(* Logix 5000 project; controller AdvManLab vendor 1 type 14 code 158 rev 28.12; software revision 28.01 *)

TASK Festo (periodic, rate 50 ms, priority 10, watchdog 50 ms) : Data_Collection
TASK MainTask (continuous, watchdog 500 ms) : MainProgram
TASK SafetyTask (periodic, rate 20 ms, priority 10, watchdog 20 ms) : SafetyProgram

MODULES
   Local : vendor 1 type 14 code 158 (ICP 0, rev 28.12)
      EN2TR03 : vendor 1 type 12 code 200 (Ethernet 192.168.1.42, ICP 3, rev 5.8)
         CNC1 : vendor 1 type 14 code 178 (Ethernet 192.168.1.110, rev 28.1, $33999264$ RPI 10 ms)
         CNC4 : vendor 1 type 14 code 178 (Ethernet 192.168.1.140, rev 28.1, $0e99d22c$ RPI 10 ms)
         CNC3 : vendor 1 type 14 code 178 (Ethernet 192.168.1.130, rev 28.1, $2d1da0b6$ RPI 10 ms)
         CNC2 : vendor 1 type 14 code 178 (Ethernet 192.168.1.120, rev 28.1, $009657be$ RPI 10 ms)
      EN2TR02 : vendor 1 type 12 code 200 (ICP 2, Ethernet 192.168.1.41, rev 5.1)
         ConvETAP_N051 : 1783-ETAP (Ethernet 192.168.1.51, rev 2.2)
              Conv_N053:3:I.0   // C2 Entry RFID2
              Conv_N053:3:I.2   // C2 exit RFID4
              Conv_N053:3:I.1   // C1 Inside RFID3
              C3_N031:5:I.1   // C3 Outside RFID6
              C3_N031:5:I.0   // C3 Inside RFID5
              C2_N021:7:O.3   // CNC2_Switch_On
              C1_N011:6:I.7   // Inside C1 RFID1
              Main_N043:3:I.0   // C1 Entry NO RFID
         MainETAP_N044 : 1783-ETAP (Ethernet 192.168.1.44, rev 2.2)
         FanucLoopVFD_N045 : PowerFlex 525-EENET (Ethernet 192.168.1.45, rev 1.3, Output RPI 20 ms)
         ABBLoopVFD_N046 : PowerFlex 525-EENET (Ethernet 192.168.1.46, rev 1.3, Output RPI 20 ms)
         RFID_N057 : vendor 1 type 139 code 6 (Ethernet 192.168.1.57, rev 1.5, Output RPI 20 ms)
         RFID_N056 : vendor 1 type 139 code 6 (Ethernet 192.168.1.56, rev 1.5, Output RPI 20 ms)
              RFID_N056:I.Channel[0].TagPresent   // RFID5
              RFID_N056:I.Channel[1].TagPresent   // RFID6
         RFID_N054 : vendor 1 type 139 code 6 (Ethernet 192.168.1.54, rev 1.5, Output RPI 20 ms)
              RFID_N054:I.Channel[0].TagPresent   // RFID1
              RFID_N054:I.Channel[1].TagPresent   // RFID2
              RFID_N054:I.Channel[0].Data[3]   // Read tag Part #
              RFID_N054:I.Channel[0].Data[4]   // Read tag Process #
              RFID_N054:O.Channel[0].Data[3]   // Write Process #?
         RFID_N055 : vendor 1 type 139 code 6 (Ethernet 192.168.1.55, rev 1.5, Output RPI 20 ms)
              RFID_N055:I.Channel[0].TagPresent   // RFID3
              RFID_N055:I.Channel[1].TagPresent   // RFID4
         Fanuc_Rbt_C1 : ETHERNET-MODULE (Ethernet 192.168.1.12, rev 1.1, Output RPI 10 ms)
              Fanuc_Rbt_C1:I.Data[0].1   // Placement of part from CNC1 to conveyor Program finished DO[2]
              Fanuc_Rbt_C1:I.Data[0].0   // Placement of part from CNC2 to conveyor Program finished DO[1]
              Fanuc_Rbt_C1:I.Data[0].10   // Cell 1 Robot is at Hold Position (CNC2) DO[11]
              Fanuc_Rbt_C1:I.Data[0].11   // Robot has completed dropping off part (CNC2) DO[12]
              Fanuc_Rbt_C1:I.Data[0].12   // Robot has completed picking up part (CNC2) DO[13]
              Fanuc_Rbt_C1:I.Data[0].13   // Robot is dropping off part (CNC2) DO[14]
              Fanuc_Rbt_C1:I.Data[0].14   // Flip Part Program running DO[15]
              Fanuc_Rbt_C1:I.Data[0].15   // Flipping Part Program is Running DO[16]
              Fanuc_Rbt_C1:I.Data[0].2   // Pick from Conveyor and Drop on CNC2 Program running DO[3]
              Fanuc_Rbt_C1:I.Data[0].3   // Pick from Conveyor and Drop on CNC1 Program running DO[4]
              Fanuc_Rbt_C1:I.Data[0].4   // Pick from CNC2 and Drop on Conveyor Program running DO[5]
              Fanuc_Rbt_C1:I.Data[0].5   // Pick from CNC1 and Drop on Conveyor Program running DO[6]
              Fanuc_Rbt_C1:I.Data[0].6   // Cell 1 Robot is at Hold Position DI[7]
              Fanuc_Rbt_C1:I.Data[0].7   // Robot has completed dropping off part DI[8]
              Fanuc_Rbt_C1:I.Data[0].8   // Robot has completed picking up part DI[9]
              Fanuc_Rbt_C1:I.Data[0].9   // Robot is dropping off part DI[10]
              Fanuc_Rbt_C1:I.Data[1].0   // Pallet with Flipped Part can be Let Go DO[17]
              Fanuc_Rbt_C1:O.Data[0].0   // Pick from Conveyor and drop on CNC 2 DI[1]
              Fanuc_Rbt_C1:O.Data[0].1   // Pick from Conveyor and drop on CNC 1 DI[2]
              Fanuc_Rbt_C1:O.Data[0].2   // Pick from CNC2 and Drop on conveyor DI[3]
              Fanuc_Rbt_C1:O.Data[0].3   // Pick from CNC1 and Drop on conveyor DI[4]
              Fanuc_Rbt_C1:O.Data[0].4   // Flip part to machine top of cabin/trunk DI[5]
              Fanuc_Rbt_C1:O.Data[0].6   // Cell 1 Robot OK to Continue DI[7]
              Fanuc_Rbt_C1:O.Data[0].7   // Cell 2 Robot OK to Continue (CNC2) DI[8]
         Fanuc_Rbt_C2 : ETHERNET-MODULE (Ethernet 192.168.1.22, rev 1.1, Output RPI 8 ms)
              Fanuc_Rbt_C2:I.Data[0].10   // Cell 2 Robot is at Hold Position (CNC3) DO[11]
              Fanuc_Rbt_C2:I.Data[0].11   // Robot has completed dropping off part (CNC3) DO[12]
              Fanuc_Rbt_C2:I.Data[0].12   // Robot has completed picking up part (CNC3) DO[13]
              Fanuc_Rbt_C2:I.Data[0].13   // Robot is dropping off part (CNC3) DO[14]
              Fanuc_Rbt_C2:I.Data[0].2   // Pick from Conveyor and Drop on CNC3 Program running DO[3]
              Fanuc_Rbt_C2:I.Data[0].3   // Pick from Conveyor and Drop on CNC4 Program running DO[4]
              Fanuc_Rbt_C2:I.Data[0].4   // Pick from CNC3 and Drop on Conveyor Program running DO[5]
              Fanuc_Rbt_C2:I.Data[0].5   // Pick from CNC4 and Drop on Conveyor Program running DO[6]
              Fanuc_Rbt_C2:I.Data[0].6   // Cell 2 Robot is at Hold Position (CNC4) DO[7]
              Fanuc_Rbt_C2:I.Data[0].7   // Robot has completed dropping off part (CNC4) DO[8]
              Fanuc_Rbt_C2:I.Data[0].8   // Robot has completed picking up part (CNC4) DO[9]
              Fanuc_Rbt_C2:I.Data[0].9   // Robot is dropping off part (CNC4) DO[10]
              Fanuc_Rbt_C2:O.Data[0].0   // Pick from Conveyor and drop on CNC 3 DI[1]
              Fanuc_Rbt_C2:O.Data[0].1   // Pick from Conveyor and drop on CNC 4 DI[2]
              Fanuc_Rbt_C2:O.Data[0].2   // Pick from CNC3 and Drop on conveyor DI[3]
              Fanuc_Rbt_C2:O.Data[0].3   // Pick from CNC4 and Drop on conveyor DI[4]
              Fanuc_Rbt_C2:O.Data[0].6   // Cell 2 Robot OK to Continue (CNC4) DI[7]
              Fanuc_Rbt_C2:O.Data[0].7   // Cell 2 Robot OK to Continue (CNC3) DI[8]
              Fanuc_Rbt_C2:O.Data[1].0   // DI[17] Start
              Fanuc_Rbt_C2:O.Data[3].0   // DI[49]
              Fanuc_Rbt_C2:O.Data[3].1   // DI[50] Cycle Start / Run
              Fanuc_Rbt_C2:O.Data[3].2   // DI[51] Continue
              Fanuc_Rbt_C2:O.Data[3].8   // GI[1/0]
         Festo_CPX : ETHERNET-MODULE (Ethernet 192.168.1.245, rev 1.1, Output RPI 10 ms)
              Festo_CPX:I.Data[0]   // #0: FB36 - (I0)-LB
              Festo_CPX:I.Data[10]   // #5: 4AI-P-D10 - (I0)-LB
              Festo_CPX:I.Data[11]   // #5: 4AI-P-D10 - (I0)-HB
              Festo_CPX:I.Data[12]   // #5: 4AI-P-D10 - (I1)-LB
              Festo_CPX:I.Data[13]   // #5: 4AI-P-D10 - (I1)-HB
              Festo_CPX:I.Data[14]   // #5: 4AI-P-D10 - (I2)-LB
              Festo_CPX:I.Data[15]   // #5: 4AI-P-D10 - (I2)-HB
              Festo_CPX:I.Data[16]   // #5: 4AI-P-D10 - (I3)-LB
              Festo_CPX:I.Data[17]   // #5: 4AI-P-D10 - (I3)-HB
              Festo_CPX:I.Data[18]   // #6: MPA(S/F)-P - (I0)-LB
              Festo_CPX:I.Data[19]   // #6: MPA(S/F)-P - (I0)-HB
              Festo_CPX:I.Data[1]   // #0: FB36 - (I0)-HB
              Festo_CPX:I.Data[20]   // #3: 16DI-D - (I0-7)
              Festo_CPX:I.Data[21]   // #3: 16DI-D - (I8-15)
              Festo_CPX:I.Data[2]   // #1: 4AI-I - (I0)-LB
              Festo_CPX:I.Data[3]   // #1: 4AI-I - (I0)-HB
              Festo_CPX:I.Data[4]   // #1: 4AI-I - (I1)-LB
              Festo_CPX:I.Data[5]   // #1: 4AI-I - (I1)-HB
              Festo_CPX:I.Data[6]   // #1: 4AI-I - (I2)-LB
              Festo_CPX:I.Data[7]   // #1: 4AI-I - (I2)-HB
              Festo_CPX:I.Data[8]   // #1: 4AI-I - (I3)-LB
              Festo_CPX:I.Data[9]   // #1: 4AI-I - (I3)-HB
              Festo_CPX:O.Data[0]   // #0: FB36 - (O1)-LB
              Festo_CPX:O.Data[10]   // #10: MPA2S-D - (O0-3)
              Festo_CPX:O.Data[1]   // #0: FB36 - (O1)-HB
              Festo_CPX:O.Data[2]   // #2: 2AO - (O0)-LB
              Festo_CPX:O.Data[3]   // #2: 2AO - (O0)-HB
              Festo_CPX:O.Data[4]   // #2: 2AO - (O1)-LB
              Festo_CPX:O.Data[5]   // #2: 2AO - (O1)-HB
              Festo_CPX:O.Data[6]   // #4: 8DO - (O0-7)
              Festo_CPX:O.Data[7]   // #7: MPA2S-D - (O0-3)
              Festo_CPX:O.Data[8]   // #8: MPA2S-D - (O0-3)
              Festo_CPX:O.Data[9]   // #9: MPA2S-D - (O0-3)
              Festo_CPX:C.Data[113].0   // -
              Festo_CPX:C.Data[144].7   // -
              Festo_CPX:C.Data[28].7   // -
              Festo_CPX:C.Data[2].7   // -
              Festo_CPX:C.Data[53].0   // -
              Festo_CPX:C.Data[53].2   // -
              Festo_CPX:C.Data[53].3   // -
              Festo_CPX:C.Data[53].4   // -
              Festo_CPX:C.Data[53].5   // -
              Festo_CPX:C.Data[53].6   // -
              Festo_CPX:C.Data[54].0   // -
              Festo_CPX:C.Data[54].2   // -
              Festo_CPX:C.Data[54].4   // -
              Festo_CPX:C.Data[113].1   // -
              Festo_CPX:C.Data[113].2   // -
              Festo_CPX:C.Data[54].5   // -
              Festo_CPX:C.Data[54].6   // -
              Festo_CPX:C.Data[54].7   // -
              Festo_CPX:C.Data[55].0   // -
              Festo_CPX:C.Data[55].1   // -
              Festo_CPX:C.Data[55].2   // -
              Festo_CPX:C.Data[55].3   // -
              Festo_CPX:C.Data[55].6   // -
              Festo_CPX:C.Data[55].7   // -
              Festo_CPX:C.Data[67].4   // -
              Festo_CPX:C.Data[67].5   // -
              Festo_CPX:C.Data[113].3   // -
              Festo_CPX:C.Data[113].4   // -
              Festo_CPX:C.Data[113].5   // -
              Festo_CPX:C.Data[1].7   // -
              Festo_CPX:C.Data[21].2   // -
              Festo_CPX:C.Data[21].3   // -
              Festo_CPX:C.Data[21].4   // -
              Festo_CPX:C.Data[21].5   // -
              Festo_CPX:C.Data[113].6   // -
              Festo_CPX:C.Data[128].1   // O0: Failsafe - Bit1
              Festo_CPX:C.Data[67].6   // -
              Festo_CPX:C.Data[67].7   // -
              Festo_CPX:C.Data[74].1   // -
              Festo_CPX:C.Data[74].2   // -
              Festo_CPX:C.Data[74].3   // -
              Festo_CPX:C.Data[74].4   // -
              Festo_CPX:C.Data[74].5   // -
              Festo_CPX:C.Data[74].6   // -
              Festo_CPX:C.Data[74].7   // -
              Festo_CPX:C.Data[75].1   // -
              Festo_CPX:C.Data[75].2   // -
              Festo_CPX:C.Data[114].2   // -
              Festo_CPX:C.Data[114].5   // -
              Festo_CPX:C.Data[75].3   // -
              Festo_CPX:C.Data[80].0   // -
              Festo_CPX:C.Data[80].3   // -
              Festo_CPX:C.Data[80].4   // -
              Festo_CPX:C.Data[80].5   // -
              Festo_CPX:C.Data[80].6   // -
              Festo_CPX:C.Data[80].7   // -
              Festo_CPX:C.Data[81].0   // -
              Festo_CPX:C.Data[81].2   // -
              Festo_CPX:C.Data[81].3   // -
              Festo_CPX:C.Data[81].4   // -
              Festo_CPX:C.Data[114].6   // -
              Festo_CPX:C.Data[114].7   // -
              Festo_CPX:C.Data[115].2   // -
              Festo_CPX:C.Data[21].6   // -
              Festo_CPX:C.Data[21].7   // -
              Festo_CPX:C.Data[26].1   // -
              Festo_CPX:C.Data[26].2   // -
              Festo_CPX:C.Data[26].3   // -
              Festo_CPX:C.Data[115].3   // -
              Festo_CPX:C.Data[115].4   // -
              Festo_CPX:C.Data[81].5   // -
              Festo_CPX:C.Data[81].6   // -
              Festo_CPX:C.Data[81].7   // -
              Festo_CPX:C.Data[87].0   // -
              Festo_CPX:C.Data[87].1   // -
              Festo_CPX:C.Data[87].2   // -
              Festo_CPX:C.Data[87].3   // -
              Festo_CPX:C.Data[87].4   // -
              Festo_CPX:C.Data[87].5   // -
              Festo_CPX:C.Data[87].6   // -
              Festo_CPX:C.Data[8].2   // -
              Festo_CPX:C.Data[115].5   // -
              Festo_CPX:C.Data[115].6   // -
              Festo_CPX:C.Data[8].3   // -
              Festo_CPX:C.Data[115].7   // -
              Festo_CPX:C.Data[26].4   // -
              Festo_CPX:C.Data[26].5   // -
              Festo_CPX:C.Data[26].6   // -
              Festo_CPX:C.Data[27].1   // -
              Festo_CPX:C.Data[27].2   // -
              Festo_CPX:C.Data[116].2   // -
              Festo_CPX:C.Data[128].2   // O1: Failsafe - Bit0
              Festo_CPX:C.Data[8].4   // -
              Festo_CPX:C.Data[8].5   // -
              Festo_CPX:C.Data[8].6   // -
              Festo_CPX:C.Data[8].7   // -
              Festo_CPX:C.Data[116].3   // -
              Festo_CPX:C.Data[116].4   // -
              Festo_CPX:C.Data[116].5   // -
              Festo_CPX:C.Data[116].6   // -
              Festo_CPX:C.Data[116].7   // -
              Festo_CPX:C.Data[27].3   // -
              Festo_CPX:C.Data[27].4   // -
              Festo_CPX:C.Data[27].5   // -
              Festo_CPX:C.Data[27].6   // -
              Festo_CPX:C.Data[27].7   // -
              Festo_CPX:C.Data[126].0   // -
              Festo_CPX:C.Data[139].5   // -
              Festo_CPX:C.Data[2].6   // System start
              Festo_CPX:C.Data[126].5   // -
              Festo_CPX:C.Data[126].1   // -
              Festo_CPX:C.Data[28].2   // -
              Festo_CPX:C.Data[139].6   // -
              Festo_CPX:C.Data[28].3   // -
              Festo_CPX:C.Data[28].4   // -
              Festo_CPX:C.Data[113]   // Monitor parameters
              Festo_CPX:C.Data[114].3   // Diagnostic Delay - Bit0
              Festo_CPX:C.Data[12].3   // Fault end filter
              Festo_CPX:C.Data[121]   // I0: Hysteresis - HB
              Festo_CPX:C.Data[138].7   // -
              Festo_CPX:C.Data[132].3   // Monitor SCV
              Festo_CPX:C.Data[100]   // I3: Lower limit - HB
              Festo_CPX:C.Data[126].4   // -
              Festo_CPX:C.Data[117]   // I0: Lower limit - HB
              Festo_CPX:C.Data[27]   // Behaviour after SCS
              Festo_CPX:C.Data[28].5   // -
              Festo_CPX:C.Data[28].6   // -
              Festo_CPX:C.Data[139].4   // -
              Festo_CPX:C.Data[126].6   // -
              Festo_CPX:C.Data[22]   // O0: Failsafe Value - HB
              Festo_CPX:C.Data[23]   // O0: Failsafe Value - LB
              Festo_CPX:C.Data[146].4   // O2: Failsafe - Bit0
              Festo_CPX:C.Data[115]   // Monitor lower limit, Monitor upper limit
              Festo_CPX:C.Data[114]   // Dimension unit, Diagnostic Delay
              Festo_CPX:C.Data[12].7   // Module/channel filter - Bit1
              Festo_CPX:C.Data[132]   // Monitor Vout/Vval, Monitor SCV
              Festo_CPX:C.Data[139].0   // O0: Monitor wire fracture
              Festo_CPX:C.Data[139].1   // O1: Monitor wire fracture
              Festo_CPX:C.Data[139].2   // O2: Monitor wire fracture
              Festo_CPX:C.Data[139].3   // O3: Monitor wire fracture
              Festo_CPX:C.Data[111]   // #6: MPA(S/F)-P - Analogue Input Press.
              Festo_CPX:C.Data[132].2   // Monitor Vout/Vval
              Festo_CPX:C.Data[123]   // #7: MPA2S-D - Pneumatic module
              Festo_CPX:C.Data[134]   // Failsafe (00=Hold, 01=Reset, 10=Set)
              Festo_CPX:C.Data[133]   // Monitor wire fracture
              Festo_CPX:C.Data[126]   // Monitor Vout/Vval, Monitor SCV
              Festo_CPX:C.Data[133].0   // O0: Monitor wire fracture
              Festo_CPX:C.Data[24]   // #1: 4AI-I - Analogue input
              Festo_CPX:C.Data[26]   // Monitor SCS, Monitor parameters
              Festo_CPX:C.Data[146].5   // O2: Failsafe - Bit1
              Festo_CPX:C.Data[146].6   // O3: Failsafe - Bit0
              Festo_CPX:C.Data[139].7   // -
              Festo_CPX:C.Data[138].2   // Monitor Vout/Vval
              Festo_CPX:C.Data[139]   // Monitor wire fracture
              Festo_CPX:C.Data[129]   // #8: MPA2S-D - Pneumatic module
              Festo_CPX:C.Data[133].1   // O1: Monitor wire fracture
              Festo_CPX:C.Data[12].1   // Run/Stop filter 2 - Bit1
              Festo_CPX:C.Data[133].2   // O2: Monitor wire fracture
              Festo_CPX:C.Data[12].2   // Run/Stop filter 2 - Bit2
              Festo_CPX:C.Data[133].3   // O3: Monitor wire fracture
              Festo_CPX:C.Data[12].4   // Fault number filter - Bit0
              Festo_CPX:C.Data[134].0   // O0: Failsafe - Bit0
              Festo_CPX:C.Data[12].5   // Fault number filter - Bit1
              Festo_CPX:C.Data[12].6   // Module/channel filter - Bit0
              Festo_CPX:C.Data[134].1   // O0: Failsafe - Bit1
              Festo_CPX:C.Data[26].7   // Monitor parameters
              Festo_CPX:C.Data[27].0   // Behaviour after SCS
              Festo_CPX:C.Data[146].7   // O3: Failsafe - Bit1
              Festo_CPX:C.Data[16]   // #0: FB36 - EtherNet/IP Remote-IO V2
              Festo_CPX:C.Data[144].0   // -
              Festo_CPX:C.Data[101]   // I3: Lower limit - LB
              Festo_CPX:C.Data[138].3   // Monitor SCV
              Festo_CPX:C.Data[105]   // I1: Upper limit - LB
              Festo_CPX:C.Data[106]   // I2: Upper limit - HB
              Festo_CPX:C.Data[126].7   // -
              Festo_CPX:C.Data[107]   // I2: Upper limit - LB
              Festo_CPX:C.Data[108]   // I3: Upper limit - HB
              Festo_CPX:C.Data[109]   // I3: Upper limit - LB
              Festo_CPX:C.Data[116]   // Filter measured value
              Festo_CPX:C.Data[110]   // Sub-module-code
              Festo_CPX:C.Data[145].5   // -
              Festo_CPX:C.Data[126].3   // Monitor SCV
              Festo_CPX:C.Data[145].6   // -
              Festo_CPX:C.Data[127].4   // -
              Festo_CPX:C.Data[114].0   // Dimension unit - Bit0
              Festo_CPX:C.Data[144].3   // Monitor SCV
              Festo_CPX:C.Data[127].5   // -
              Festo_CPX:C.Data[14]   // Channel number
              Festo_CPX:C.Data[2].0   // Fail safe - Bit0
              Festo_CPX:C.Data[145].7   // -
              Festo_CPX:C.Data[127].6   // -
              Festo_CPX:C.Data[102]   // I0: Upper limit - HB
              Festo_CPX:C.Data[103]   // I0: Upper limit - LB
              Festo_CPX:C.Data[33].0   // I0: Signal range - Bit0
              Festo_CPX:C.Data[2].4   // Idle mode - Bit0
              Festo_CPX:C.Data[58]   // Signal range
              Festo_CPX:C.Data[30]   // I1: Diagnostic functions
              Festo_CPX:C.Data[114].4   // Diagnostic Delay - Bit1
              Festo_CPX:C.Data[49]   // I3: Upper limit - HB
              Festo_CPX:C.Data[70]   // O1: Failsafe Value - HB
              Festo_CPX:C.Data[59]   // O0: Lower limit - HB
              Festo_CPX:C.Data[67]   // Failsafe (00=Hold, 01=Value)
              Festo_CPX:C.Data[41]   // I3: Lower limit - HB
              Festo_CPX:C.Data[75]   // Behaviour after SCS, Input debounce time, Signal extension time
              Festo_CPX:C.Data[28].0   // Input format - Bit0
              Festo_CPX:C.Data[28].1   // Input format - Bit1
              Festo_CPX:C.Data[40]   // I2: Lower limit - LB
              Festo_CPX:C.Data[31]   // I2: Diagnostic functions
              Festo_CPX:C.Data[80]   // Monitor SCO (Output/Actuator Supply), Monitor Vout/Vval
              Festo_CPX:C.Data[33].3   // I1: Signal range - Bit1
              Festo_CPX:C.Data[66]   // O1: Upper limit - LB
              Festo_CPX:C.Data[134].2   // O1: Failsafe - Bit0
              Festo_CPX:C.Data[61]   // O1: Lower limit - HB
              Festo_CPX:C.Data[60]   // O0: Lower limit - LB
              Festo_CPX:C.Data[58].2   // O0: Signal range - Bit2
              Festo_CPX:C.Data[115].0   // I0: Monitor lower limit
              Festo_CPX:C.Data[54].1   // Behaviour after SCO (Output/Actuator Supply)
              Festo_CPX:C.Data[56]   // O0: Diagnostic functions
              Festo_CPX:C.Data[54]   // Behaviour after SCO (Output/Actuator Supply), Behaviour after SCA (analogue signal)
              Festo_CPX:C.Data[75].5   // Input debounce time - Bit1
              Festo_CPX:C.Data[68]   // O0: Failsafe Value - HB
              Festo_CPX:C.Data[64]   // O0: Upper limit - LB
              Festo_CPX:C.Data[58].3   // O0: Signal range - Bit3
              Festo_CPX:C.Data[67].0   // O0: Failsafe - Bit0
              Festo_CPX:C.Data[75].6   // Signal extension time - Bit0
              Festo_CPX:C.Data[62]   // O1: Lower limit - LB
              Festo_CPX:C.Data[88]   // Dimension unit, Pressure difference calc. Ch0-1, Pressure difference calc. Ch2-3, Monitor sensor limit Ch0, Monitor sensor limit Ch1, Monitor sensor limit Ch2, Monitor sensor limit Ch3
              Festo_CPX:C.Data[58].6   // O1: Signal range - Bit2
              Festo_CPX:C.Data[12]   // Run/Stop filter 2, Fault end filter, Fault number filter, Module/channel filter
              Festo_CPX:C.Data[69]   // O0: Failsafe Value - LB
              Festo_CPX:C.Data[58].4   // O1: Signal range - Bit0
              Festo_CPX:C.Data[58].7   // O1: Signal range - Bit3
              Festo_CPX:C.Data[58].1   // O0: Signal range - Bit1
              Festo_CPX:C.Data[71]   // O1: Failsafe Value - LB
              Festo_CPX:C.Data[67].1   // O0: Failsafe - Bit1
              Festo_CPX:C.Data[75].4   // Input debounce time - Bit0
              Festo_CPX:C.Data[67].2   // O1: Failsafe - Bit0
              Festo_CPX:C.Data[32]   // I3: Diagnostic functions
              Festo_CPX:C.Data[57]   // O1: Diagnostic functions
              Festo_CPX:C.Data[58].5   // O1: Signal range - Bit1
              Festo_CPX:C.Data[65]   // O1: Upper limit - HB
              Festo_CPX:C.Data[55].5   // Output format - Bit1
              Festo_CPX:C.Data[29]   // I0: Diagnostic functions
              Festo_CPX:C.Data[72]   // #3: 16DI-D - Input module
              Festo_CPX:C.Data[145].3   // O3: Monitor wire fracture
              Festo_CPX:C.Data[33].1   // I0: Signal range - Bit1
              Festo_CPX:C.Data[42]   // I3: Lower limit - LB
              Festo_CPX:C.Data[53].1   // Monitor SCO (Output/Actuator Supply)
              Festo_CPX:C.Data[54].3   // Behaviour after SCA (analogue signal)
              Festo_CPX:C.Data[55].4   // Output format - Bit0
              Festo_CPX:C.Data[1].5   // -
              Festo_CPX:C.Data[1].6   // -
              Festo_CPX:C.Data[15]   // Fault number
              Festo_CPX:C.Data[140].6   // O3: Failsafe - Bit0
              Festo_CPX:C.Data[128].3   // O1: Failsafe - Bit1
              Festo_CPX:C.Data[35]   // I0: Lower limit - HB
              Festo_CPX:C.Data[127].7   // -
              Festo_CPX:C.Data[1]   // Diagnosis
              Festo_CPX:C.Data[114].1   // Dimension unit - Bit1
              Festo_CPX:C.Data[104]   // I1: Upper limit - HB
              Festo_CPX:C.Data[115].1   // I0: Monitor upper limit
              Festo_CPX:C.Data[33].4   // I2: Signal range - Bit0
              Festo_CPX:C.Data[127].0   // O0: Monitor wire fracture
              Festo_CPX:C.Data[140].1   // O0: Failsafe - Bit1
              Festo_CPX:C.Data[33].5   // I2: Signal range - Bit1
              Festo_CPX:C.Data[50]   // I3: Upper limit - LB
              Festo_CPX:C.Data[51]   // #2: 2AO - Analogue output
              Festo_CPX:C.Data[53]   // Monitor SCO (Output/Actuator Supply), Monitor parameters
              Festo_CPX:C.Data[127].1   // O1: Monitor wire fracture
              Festo_CPX:C.Data[127].2   // O2: Monitor wire fracture
              Festo_CPX:C.Data[127].3   // O3: Monitor wire fracture
              Festo_CPX:C.Data[33].6   // I3: Signal range - Bit0
              Festo_CPX:C.Data[33].7   // I3: Signal range - Bit1
              Festo_CPX:C.Data[34]   // Filter measured value
              Festo_CPX:C.Data[134].3   // O1: Failsafe - Bit1
              Festo_CPX:C.Data[134].4   // O2: Failsafe - Bit0
              Festo_CPX:C.Data[134].5   // O2: Failsafe - Bit1
              Festo_CPX:C.Data[34].0   // I0: Filter measured value - Bit0
              Festo_CPX:C.Data[34].1   // I0: Filter measured value - Bit1
              Festo_CPX:C.Data[144].2   // Monitor Vout/Vval
              Festo_CPX:C.Data[128].4   // O2: Failsafe - Bit0
              Festo_CPX:C.Data[128].5   // O2: Failsafe - Bit1
              Festo_CPX:C.Data[128].6   // O3: Failsafe - Bit0
              Festo_CPX:C.Data[140].2   // O1: Failsafe - Bit0
              Festo_CPX:C.Data[140].3   // O1: Failsafe - Bit1
              Festo_CPX:C.Data[140].4   // O2: Failsafe - Bit0
              Festo_CPX:C.Data[33].2   // I1: Signal range - Bit0
              Festo_CPX:C.Data[128].7   // O3: Failsafe - Bit1
              Festo_CPX:C.Data[12].0   // Run/Stop filter 2 - Bit0
              Festo_CPX:C.Data[140].7   // O3: Failsafe - Bit1
              Festo_CPX:C.Data[36]   // I0: Lower limit - LB
              Festo_CPX:C.Data[43]   // I0: Upper limit - HB
              Festo_CPX:C.Data[44]   // I0: Upper limit - LB
              Festo_CPX:C.Data[45]   // I1: Upper limit - HB
              Festo_CPX:C.Data[38]   // I1: Lower limit - LB
              Festo_CPX:C.Data[116].0   // I0: Filter measured value - Bit0
              Festo_CPX:C.Data[140]   // Failsafe (00=Hold, 01=Reset, 10=Set)
              Festo_CPX:C.Data[63]   // O0: Upper limit - HB
              Festo_CPX:C.Data[34].2   // I1: Filter measured value - Bit0
              Festo_CPX:C.Data[67].3   // O1: Failsafe - Bit1
              Festo_CPX:C.Data[140].0   // O0: Failsafe - Bit0
              Festo_CPX:C.Data[21]   // Failsafe (00=Hold, 01=Value)
              Festo_CPX:C.Data[145]   // Monitor wire fracture
              Festo_CPX:C.Data[116].1   // I0: Filter measured value - Bit1
              Festo_CPX:C.Data[141]   // #10: MPA2S-D - Pneumatic module
              Festo_CPX:C.Data[146]   // Failsafe (00=Hold, 01=Reset, 10=Set)
              Festo_CPX:C.Data[146].0   // O0: Failsafe - Bit0
              Festo_CPX:C.Data[145].0   // O0: Monitor wire fracture
              Festo_CPX:C.Data[146].1   // O0: Failsafe - Bit1
              Festo_CPX:C.Data[146].2   // O1: Failsafe - Bit0
              Festo_CPX:C.Data[145].1   // O1: Monitor wire fracture
              Festo_CPX:C.Data[145].2   // O2: Monitor wire fracture
              Festo_CPX:C.Data[34].3   // I1: Filter measured value - Bit1
              Festo_CPX:C.Data[146].3   // O1: Failsafe - Bit1
              Festo_CPX:C.Data[39]   // I2: Lower limit - HB
              Festo_CPX:C.Data[37]   // I1: Lower limit - HB
              Festo_CPX:C.Data[144]   // Monitor Vout/Vval, Monitor SCV
              Festo_CPX:C.Data[2]   // CPX System Settings
              Festo_CPX:C.Data[21].0   // O0: Failsafe - Bit0
              Festo_CPX:C.Data[132].0   // -
              Festo_CPX:C.Data[46]   // I1: Upper limit - LB
              Festo_CPX:C.Data[47]   // I2: Upper limit - HB
              Festo_CPX:C.Data[48]   // I2: Upper limit - LB
              Festo_CPX:C.Data[20]   // Startup
              Festo_CPX:C.Data[122]   // I0: Hysteresis - LB
              Festo_CPX:C.Data[1].2   // Monitor Vout
              Festo_CPX:C.Data[34].4   // I2: Filter measured value - Bit0
              Festo_CPX:C.Data[134].6   // O3: Failsafe - Bit0
              Festo_CPX:C.Data[34].5   // I2: Filter measured value - Bit1
              Festo_CPX:C.Data[134].7   // O3: Failsafe - Bit1
              Festo_CPX:C.Data[34].6   // I3: Filter measured value - Bit0
              Festo_CPX:C.Data[135]   // #9: MPA2S-D - Pneumatic module
              Festo_CPX:C.Data[34].7   // I3: Filter measured value - Bit1
              Festo_CPX:C.Data[138]   // Monitor Vout/Vval, Monitor SCV
              Festo_CPX:C.Data[2].5   // Idle mode - Bit1
              Festo_CPX:C.Data[127]   // Monitor wire fracture
              Festo_CPX:C.Data[128]   // Failsafe (00=Hold, 01=Reset, 10=Set)
              Festo_CPX:C.Data[126].2   // Monitor Vout/Vval
              Festo_CPX:C.Data[53].7   // Monitor parameters
              Festo_CPX:C.Data[58].0   // O0: Signal range - Bit0
              Festo_CPX:C.Data[132].1   // -
              Festo_CPX:C.Data[140].5   // O2: Failsafe - Bit1
              Festo_CPX:C.Data[21].1   // O0: Failsafe - Bit1
              Festo_CPX:C.Data[128].0   // O0: Failsafe - Bit0
              Festo_CPX:C.Data[113].7   // Monitor parameters
              Festo_CPX:C.Data[118]   // I0: Lower limit - LB
              Festo_CPX:C.Data[2].1   // Fail safe - Bit1
              Festo_CPX:C.Data[2].2   // Force mode - Bit0
              Festo_CPX:C.Data[13]   // Module number
              Festo_CPX:C.Data[1].1   // Monitor SCO
              Festo_CPX:C.Data[132].4   // -
              Festo_CPX:C.Data[132].5   // -
              Festo_CPX:C.Data[132].6   // -
              Festo_CPX:C.Data[132].7   // -
              Festo_CPX:C.Data[144].1   // -
              Festo_CPX:C.Data[144].4   // -
              Festo_CPX:C.Data[144].5   // -
              Festo_CPX:C.Data[144].6   // -
              Festo_CPX:C.Data[133].4   // -
              Festo_CPX:C.Data[133].5   // -
              Festo_CPX:C.Data[133].6   // -
              Festo_CPX:C.Data[133].7   // -
              Festo_CPX:C.Data[138].0   // -
              Festo_CPX:C.Data[138].1   // -
              Festo_CPX:C.Data[138].4   // -
              Festo_CPX:C.Data[138].5   // -
              Festo_CPX:C.Data[33]   // Signal range
              Festo_CPX:C.Data[55]   // Output format
              Festo_CPX:C.Data[145].4   // -
              Festo_CPX:C.Data[138].6   // -
              Festo_CPX:C.Data[2].3   // Force mode - Bit1
              Festo_CPX:C.Data[1].3   // Monitor Vval
              Festo_CPX:C.Data[1].0   // Monitor SCS
              Festo_CPX:C.Data[28]   // Input format
              Festo_CPX:C.Data[119]   // I0: Upper limit - HB
              Festo_CPX:C.Data[120]   // I0: Upper limit - LB
              Festo_CPX:C.Data[1].4   // Monitor SCV
              Festo_CPX:C.Data[26].0   // Monitor SCS
              Festo_CPX:C.Data[74]   // Monitor SCS
              Festo_CPX:C.Data[74].0   // Monitor SCS
              Festo_CPX:C.Data[75].0   // Behaviour after SCS
              Festo_CPX:C.Data[75].7   // Signal extension time - Bit1
              Festo_CPX:C.Data[76]   // Signal extension
              Festo_CPX:C.Data[76].0   // I0: Signal extension
              Festo_CPX:C.Data[76].1   // I1: Signal extension
              Festo_CPX:C.Data[76].2   // I2: Signal extension
              Festo_CPX:C.Data[76].3   // I3: Signal extension
              Festo_CPX:C.Data[76].4   // I4: Signal extension
              Festo_CPX:C.Data[76].5   // I5: Signal extension
              Festo_CPX:C.Data[76].6   // I6: Signal extension
              Festo_CPX:C.Data[76].7   // I7: Signal extension
              Festo_CPX:C.Data[77]   // Signal extension
              Festo_CPX:C.Data[77].0   // I8: Signal extension
              Festo_CPX:C.Data[77].1   // I9: Signal extension
              Festo_CPX:C.Data[77].2   // I10: Signal extension
              Festo_CPX:C.Data[77].3   // I11: Signal extension
              Festo_CPX:C.Data[77].4   // I12: Signal extension
              Festo_CPX:C.Data[77].5   // I13: Signal extension
              Festo_CPX:C.Data[77].6   // I14: Signal extension
              Festo_CPX:C.Data[77].7   // I15: Signal extension
              Festo_CPX:C.Data[78]   // #4: 8DO - Output module
              Festo_CPX:C.Data[80].1   // Monitor SCO (Output/Actuator Supply)
              Festo_CPX:C.Data[80].2   // Monitor Vout/Vval
              Festo_CPX:C.Data[81]   // Behaviour after SCO (Output/Actuator Supply)
              Festo_CPX:C.Data[81].1   // Behaviour after SCO (Output/Actuator Supply)
              Festo_CPX:C.Data[82]   // Failsafe (00=Hold, 01=Reset, 10=Set)
              Festo_CPX:C.Data[82].0   // O0: Failsafe - Bit0
              Festo_CPX:C.Data[82].1   // O0: Failsafe - Bit1
              Festo_CPX:C.Data[82].2   // O1: Failsafe - Bit0
              Festo_CPX:C.Data[82].3   // O1: Failsafe - Bit1
              Festo_CPX:C.Data[82].4   // O2: Failsafe - Bit0
              Festo_CPX:C.Data[82].5   // O2: Failsafe - Bit1
              Festo_CPX:C.Data[82].6   // O3: Failsafe - Bit0
              Festo_CPX:C.Data[82].7   // O3: Failsafe - Bit1
              Festo_CPX:C.Data[83]   // Failsafe (00=Hold, 01=Reset, 10=Set)
              Festo_CPX:C.Data[83].0   // O4: Failsafe - Bit0
              Festo_CPX:C.Data[83].1   // O4: Failsafe - Bit1
              Festo_CPX:C.Data[83].2   // O5: Failsafe - Bit0
              Festo_CPX:C.Data[83].3   // O5: Failsafe - Bit1
              Festo_CPX:C.Data[83].4   // O6: Failsafe - Bit0
              Festo_CPX:C.Data[83].5   // O6: Failsafe - Bit1
              Festo_CPX:C.Data[83].6   // O7: Failsafe - Bit0
              Festo_CPX:C.Data[83].7   // O7: Failsafe - Bit1
              Festo_CPX:C.Data[84]   // #5: 4AI-P-D10 - Analogue input press.
              Festo_CPX:C.Data[87]   // Monitor parameters
              Festo_CPX:C.Data[87].7   // Monitor parameters
              Festo_CPX:C.Data[88].0   // Dimension unit - Bit0
              Festo_CPX:C.Data[88].1   // Dimension unit - Bit1
              Festo_CPX:C.Data[88].2   // Pressure difference calc. Ch0-1
              Festo_CPX:C.Data[88].3   // Pressure difference calc. Ch2-3
              Festo_CPX:C.Data[88].4   // Monitor sensor limit Ch0
              Festo_CPX:C.Data[88].5   // Monitor sensor limit Ch1
              Festo_CPX:C.Data[88].6   // Monitor sensor limit Ch2
              Festo_CPX:C.Data[88].7   // Monitor sensor limit Ch3
              Festo_CPX:C.Data[89]   // Hystereses - HB
              Festo_CPX:C.Data[8]   // Trace Parameters
              Festo_CPX:C.Data[8].0   // Entries remanent at Power On
              Festo_CPX:C.Data[8].1   // Run/Stop filter 1
              Festo_CPX:C.Data[90]   // Hystereses - LB
              Festo_CPX:C.Data[91]   // Filter measured value
              Festo_CPX:C.Data[91].0   // I0: Filter measured value - Bit0
              Festo_CPX:C.Data[91].1   // I0: Filter measured value - Bit1
              Festo_CPX:C.Data[91].2   // I1: Filter measured value - Bit0
              Festo_CPX:C.Data[91].3   // I1: Filter measured value - Bit1
              Festo_CPX:C.Data[91].4   // I2: Filter measured value - Bit0
              Festo_CPX:C.Data[91].5   // I2: Filter measured value - Bit1
              Festo_CPX:C.Data[91].6   // I3: Filter measured value - Bit0
              Festo_CPX:C.Data[91].7   // I3: Filter measured value - Bit1
              Festo_CPX:C.Data[92]   // Diagnostic Delay
              Festo_CPX:C.Data[92].0   // I0: Diagnostic Delay - Bit0
              Festo_CPX:C.Data[92].1   // I0: Diagnostic Delay - Bit1
              Festo_CPX:C.Data[92].2   // I1: Diagnostic Delay - Bit0
              Festo_CPX:C.Data[92].3   // I1: Diagnostic Delay - Bit1
              Festo_CPX:C.Data[92].4   // I2: Diagnostic Delay - Bit0
              Festo_CPX:C.Data[92].5   // I2: Diagnostic Delay - Bit1
              Festo_CPX:C.Data[92].6   // I3: Diagnostic Delay - Bit0
              Festo_CPX:C.Data[92].7   // I3: Diagnostic Delay - Bit1
              Festo_CPX:C.Data[93]   // Monitor - lower limit, Monitor - upper limit
              Festo_CPX:C.Data[93].0   // I0: Monitor - lower limit
              Festo_CPX:C.Data[93].1   // I0: Monitor - upper limit
              Festo_CPX:C.Data[93].2   // I1: Monitor - lower limit
              Festo_CPX:C.Data[93].3   // I1: Monitor - upper limit
              Festo_CPX:C.Data[93].4   // I2: Monitor - lower limit
              Festo_CPX:C.Data[93].5   // I2: Monitor - upper limit
              Festo_CPX:C.Data[93].6   // I3: Monitor - lower limit
              Festo_CPX:C.Data[93].7   // I3: Monitor - upper limit
              Festo_CPX:C.Data[94]   // I0: Lower limit - HB
              Festo_CPX:C.Data[95]   // I0: Lower limit - LB
              Festo_CPX:C.Data[96]   // I1: Lower limit - HB
              Festo_CPX:C.Data[97]   // I1: Lower limit - LB
              Festo_CPX:C.Data[98]   // I2: Lower limit - HB
              Festo_CPX:C.Data[99]   // I2: Lower limit - LB
         NI_1752_1 : ETHERNET-MODULE (Ethernet 192.168.1.100, rev 1.1, Output RPI 10 ms)
              NI_1752_1:I.Data   // VBAI:
              NI_1752_1:I.Data[0]   // BOOL 0-31 (0-7 Reserved by VBAI)
              NI_1752_1:I.Data[10]   // DINT 0
              NI_1752_1:I.Data[11]   // DINT 1
              NI_1752_1:I.Data[12]   // DINT 2
              NI_1752_1:I.Data[13]   // DINT 3
              NI_1752_1:I.Data[14]   // DINT 4
              NI_1752_1:I.Data[15]   // DINT 5
              NI_1752_1:I.Data[16]   // DINT 6
              NI_1752_1:I.Data[17]   // DINT 7
              NI_1752_1:I.Data[18]   // DINT 8
              NI_1752_1:I.Data[19]   // DINT 9
              NI_1752_1:I.Data[1]   // SINT 0-3
              NI_1752_1:I.Data[20]   // DINT 10
              NI_1752_1:I.Data[21]   // DINT 11
              NI_1752_1:I.Data[22]   // REAL 0
              NI_1752_1:I.Data[23]   // REAL 1
              NI_1752_1:I.Data[24]   // REAL 2
              NI_1752_1:I.Data[25]   // REAL 3
              NI_1752_1:I.Data[26]   // REAL 4
              NI_1752_1:I.Data[27]   // REAL 5
              NI_1752_1:I.Data[28]   // REAL 6
              NI_1752_1:I.Data[29]   // REAL 7
              NI_1752_1:I.Data[2]   // SINT 4-7
              NI_1752_1:I.Data[30]   // REAL 8
              NI_1752_1:I.Data[31]   // REAL 9
              NI_1752_1:I.Data[32]   // REAL 10
              NI_1752_1:I.Data[33]   // REAL 11
              NI_1752_1:I.Data[3]   // SINT 8-11
              NI_1752_1:I.Data[4]   // INT 0-1
              NI_1752_1:I.Data[5]   // INT 2-3
              NI_1752_1:I.Data[6]   // INT 4-5
              NI_1752_1:I.Data[7]   // INT 6-7
              NI_1752_1:I.Data[8]   // INT 8-9
              NI_1752_1:I.Data[9]   // INT 10-11
              NI_1752_1:O.Data   // VBAI:
              NI_1752_1:O.Data[0]   // Bool 0-31
              NI_1752_1:O.Data[10]   // DINT 0
              NI_1752_1:O.Data[11]   // DINT 1
              NI_1752_1:O.Data[12]   // DINT 2
              NI_1752_1:O.Data[13]   // DINT 3
              NI_1752_1:O.Data[14]   // DINT 4
              NI_1752_1:O.Data[15]   // DINT 5
              NI_1752_1:O.Data[16]   // DINT 6
              NI_1752_1:O.Data[17]   // DINT 7
              NI_1752_1:O.Data[18]   // DINT 8
              NI_1752_1:O.Data[19]   // DINT 9
              NI_1752_1:O.Data[1]   // SINT 0-3
              NI_1752_1:O.Data[20]   // DINT 10
              NI_1752_1:O.Data[21]   // DINT 11
              NI_1752_1:O.Data[2]   // Sint 4-7
              NI_1752_1:O.Data[3]   // Sint 8-11
              NI_1752_1:O.Data[4]   // Int 0-1
              NI_1752_1:O.Data[5]   // Int 2-3
              NI_1752_1:O.Data[6]   // Int 4-5
              NI_1752_1:O.Data[7]   // Int 6-7
              NI_1752_1:O.Data[8]   // Int 8-9
              NI_1752_1:O.Data[9]   // Int 10-11
         NI_1752_2 : ETHERNET-MODULE (Ethernet 192.168.1.101, rev 1.1, Output RPI 10 ms)   // Second NI_1752 camera
              NI_1752_2:I.Data   // VBAI:
              NI_1752_2:I.Data[0]   // BOOL 0-31 (0-7 Reserved by VBAI)
              NI_1752_2:I.Data[10]   // DINT 0
              NI_1752_2:I.Data[11]   // DINT 1
              NI_1752_2:I.Data[12]   // DINT 2
              NI_1752_2:I.Data[13]   // DINT 3
              NI_1752_2:I.Data[14]   // DINT 4
              NI_1752_2:I.Data[15]   // DINT 5
              NI_1752_2:I.Data[16]   // DINT 6
              NI_1752_2:I.Data[17]   // DINT 7
              NI_1752_2:I.Data[18]   // DINT 8
              NI_1752_2:I.Data[19]   // DINT 9
              NI_1752_2:I.Data[1]   // SINT 0-3
              NI_1752_2:I.Data[20]   // DINT 10
              NI_1752_2:I.Data[21]   // DINT 11
              NI_1752_2:I.Data[22]   // REAL 0
              NI_1752_2:I.Data[23]   // REAL 1
              NI_1752_2:I.Data[24]   // REAL 2
              NI_1752_2:I.Data[25]   // REAL 3
              NI_1752_2:I.Data[26]   // REAL 4
              NI_1752_2:I.Data[27]   // REAL 5
              NI_1752_2:I.Data[28]   // REAL 6
              NI_1752_2:I.Data[29]   // REAL 7
              NI_1752_2:I.Data[2]   // SINT 4-7
              NI_1752_2:I.Data[30]   // REAL 8
              NI_1752_2:I.Data[31]   // REAL 9
              NI_1752_2:I.Data[32]   // REAL 10
              NI_1752_2:I.Data[33]   // REAL 11
              NI_1752_2:I.Data[3]   // SINT 8-11
              NI_1752_2:I.Data[4]   // INT 0-1
              NI_1752_2:I.Data[5]   // INT 2-3
              NI_1752_2:I.Data[6]   // INT 4-5
              NI_1752_2:I.Data[7]   // INT 6-7
              NI_1752_2:I.Data[8]   // INT 8-9
              NI_1752_2:I.Data[9]   // INT 10-11
              NI_1752_2:O.Data   // VBAI:
              NI_1752_2:O.Data[10]   // DINT 0
              NI_1752_2:O.Data[11]   // DINT 1
              NI_1752_2:O.Data[12]   // DINT 2
              NI_1752_2:O.Data[13]   // DINT 3
              NI_1752_2:O.Data[14]   // DINT 4
              NI_1752_2:O.Data[15]   // DINT 5
              NI_1752_2:O.Data[16]   // DINT 6
              NI_1752_2:O.Data[17]   // DINT 7
              NI_1752_2:O.Data[18]   // DINT 8
              NI_1752_2:O.Data[19]   // DINT 9
              NI_1752_2:O.Data[1]   // SINT 0-3
              NI_1752_2:O.Data[22]   // REAL 0
              NI_1752_2:O.Data[23]   // REAL 1
              NI_1752_2:O.Data[24]   // REAL 2
              NI_1752_2:O.Data[25]   // REAL 3
              NI_1752_2:O.Data[26]   // REAL 4
              NI_1752_2:O.Data[27]   // REAL 5
              NI_1752_2:O.Data[28]   // REAL 6
              NI_1752_2:O.Data[29]   // REAL 7
              NI_1752_2:O.Data[2]   // SINT 4-7
              NI_1752_2:O.Data[30]   // REAL 8
              NI_1752_2:O.Data[31]   // REAL 9
              NI_1752_2:O.Data[4]   // INT 0-1
              NI_1752_2:O.Data[5]   // INT 2-3
              NI_1752_2:O.Data[6]   // INT 4-5
              NI_1752_2:O.Data[7]   // INT 6-7
              NI_1752_2:O.Data[0]   // Bool 0-31
              NI_1752_2:O.Data[0].0   // BOOL 0-31
              NI_1752_2:O.Data[20]   // DINT 10
              NI_1752_2:O.Data[21]   // DINT 11
              NI_1752_2:O.Data[32]   // REAL 10
              NI_1752_2:O.Data[33]   // REAL 11
              NI_1752_2:O.Data[3]   // SINT 8-11
              NI_1752_2:O.Data[8]   // INT 8-9
              NI_1752_2:O.Data[9]   // INT 10-11
         Festo_Man : vendor 26 type 12 code 14026 (Ethernet 192.168.1.70, rev 1.12, StandardDataDriven RPI 10 ms)
              Festo_Man:I1.Data[20].0   // Horozontal Retracted PPX
              Festo_Man:I1.Data[20].2   // Horozontal Mid-Point PPX
              Festo_Man:I1.Data[20].4   // Horozontal Extended PPX
              Festo_Man:I1.Data[20].6   // Vertical Raised PPX
              Festo_Man:I1.Data[20].7   // Vertical Lowered PPX
              Festo_Man:I1.Data[0]   // #0: FB36 - (I0)-LB
              Festo_Man:I1.Data[1]   // #0: FB36 - (I0)-HB
              Festo_Man:I1.Data[2]   // #1: 4AI-I - (I0)-LB
              Festo_Man:I1.Data[3]   // #1: 4AI-I - (I0)-HB
              Festo_Man:I1.Data[4]   // #1: 4AI-I - (I1)-LB
              Festo_Man:I1.Data[5]   // #1: 4AI-I - (I1)-HB
              Festo_Man:I1.Data[6]   // #1: 4AI-I - (I2)-LB
              Festo_Man:I1.Data[7]   // #1: 4AI-I - (I2)-HB
              Festo_Man:I1.Data[8]   // #1: 4AI-I - (I3)-LB
              Festo_Man:I1.Data[9]   // #1: 4AI-I - (I3)-HB
              Festo_Man:I1.Data[10]   // #5: 4AI-P-D10 - (I0)-LB
              Festo_Man:I1.Data[11]   // #5: 4AI-P-D10 - (I0)-HB
              Festo_Man:I1.Data[12]   // #5: 4AI-P-D10 - (I1)-LB
              Festo_Man:I1.Data[13]   // #5: 4AI-P-D10 - (I1)-HB
              Festo_Man:I1.Data[14]   // #5: 4AI-P-D10 - (I2)-LB
              Festo_Man:I1.Data[15]   // #5: 4AI-P-D10 - (I2)-HB
              Festo_Man:I1.Data[16]   // #5: 4AI-P-D10 - (I3)-LB
              Festo_Man:I1.Data[17]   // #5: 4AI-P-D10 - (I3)-HB
              Festo_Man:I1.Data[18]   // #6: MPA(S/F)-P - (I0)-LB
              Festo_Man:I1.Data[19]   // #6: MPA(S/F)-P - (I0)-HB
              Festo_Man:I1.Data[20]   // #3: 16DI-D - (I0-7)
              Festo_Man:I1.Data[21]   // #3: 16DI-D - (I8-15)
              Festo_Man:O1.Data[10].2   // Not Present
              Festo_Man:O1.Data[10].3   // Not Present
              Festo_Man:O1.Data[10].4   // Unused
              Festo_Man:O1.Data[10].5   // Unused
              Festo_Man:O1.Data[10].6   // Unused
              Festo_Man:O1.Data[10].7   // Unused
              Festo_Man:O1.Data[6].0   // Air On
              Festo_Man:O1.Data[7].0   // Advance Horozontal
              Festo_Man:O1.Data[7].1   // Retract Horozontal
              Festo_Man:O1.Data[7].2   // Extend Stop
              Festo_Man:O1.Data[7].3   // Do Not Use 10/18/2017
              Festo_Man:O1.Data[7].4   // Unused
              Festo_Man:O1.Data[7].5   // Unused
              Festo_Man:O1.Data[7].6   // Unused
              Festo_Man:O1.Data[7].7   // Unused
              Festo_Man:O1.Data[8].0   // Raise Vertical
              Festo_Man:O1.Data[8].1   // Lower Vertical
              Festo_Man:O1.Data[8].2   // Vacuum On
              Festo_Man:O1.Data[8].3   // Unused
              Festo_Man:O1.Data[8].4   // Unused
              Festo_Man:O1.Data[8].5   // Unused
              Festo_Man:O1.Data[8].6   // Unused
              Festo_Man:O1.Data[8].7   // Unused
              Festo_Man:O1.Data[9].0   // Suction Cup to Line
              Festo_Man:O1.Data[9].1   // Clamp to line
              Festo_Man:O1.Data[9].2   // Close Clamp
              Festo_Man:O1.Data[9].3   // Open Clamp
              Festo_Man:O1.Data[9].4   // Unused
              Festo_Man:O1.Data[9].5   // Unused
              Festo_Man:O1.Data[9].6   // Unused
              Festo_Man:O1.Data[9].7   // Unused
              Festo_Man:O1.Data[0]   // #0: FB36 - (O1)-LB
              Festo_Man:O1.Data[1]   // #0: FB36 - (O1)-HB
              Festo_Man:O1.Data[2]   // #2: 2AO - (O0)-LB
              Festo_Man:O1.Data[3]   // #2: 2AO - (O0)-HB
              Festo_Man:O1.Data[4]   // #2: 2AO - (O1)-LB
              Festo_Man:O1.Data[5]   // #2: 2AO - (O1)-HB
              Festo_Man:O1.Data[6]   // #4: 8DO - (O0-7)
              Festo_Man:O1.Data[7]   // #7: MPA2S-D - (O0-3)
              Festo_Man:O1.Data[8]   // #8: MPA2S-D - (O0-3)
              Festo_Man:O1.Data[9]   // #9: MPA2S-D - (O0-3)
              Festo_Man:O1.Data[10]   // #10: MPA2S-D - (O0-3)
              Festo_Man:O1.Data[10].1   // Not Present
              Festo_Man:O1.Data[10].0   // Not Present
         ABB_Rbt_C3 : vendor 75 type 12 code 28 (Ethernet 192.168.1.32, rev 2.5, StandardDataDriven RPI 10 ms)
         Main_N043 : 1734-AENTR (Ethernet 192.168.1.43, rev 4.1, Output RPI 20 ms)
            MainSL03 : 1734-IB8 (PointIO 3, rev 3.1)
            MainSL04 : 1734-OB8E (PointIO 4, rev 3.1)
            MainSL01 : vendor 1 type 35 code 15 (PointIO 1, rev 1.2, Input RPI 10 ms, Output RPI 20 ms)
            MainSL02 : vendor 1 type 35 code 16 (PointIO 2, rev 1.1, Input RPI 10 ms, Output RPI 20 ms)
         C1_N011 : 1734-AENTR (Ethernet 192.168.1.11, rev 4.3, Output RPI 20 ms)
            C1SL06 : 1734-IB8 (PointIO 6, rev 3.1)
            C1SL07 : 1734-OB8E (PointIO 7, rev 3.1)
            C1SL03 : vendor 1 type 35 code 15 (PointIO 3, rev 1.2, Input RPI 10 ms, Output RPI 20 ms)
            C1SL04 : vendor 1 type 35 code 15 (PointIO 4, rev 1.2, Input RPI 10 ms, Output RPI 20 ms)
            C1SL05 : vendor 1 type 35 code 16 (PointIO 5, rev 1.1, Input RPI 10 ms, Output RPI 20 ms)
            C1SL01 : vendor 1 type 35 code 15 (PointIO 1, rev 1.2, Input RPI 10 ms, Output RPI 20 ms)
            C1SL02 : vendor 1 type 35 code 15 (PointIO 2, rev 1.2, Input RPI 10 ms, Output RPI 20 ms)
         Manifold_N058 : 1734-AENTR (Ethernet 192.168.1.58, rev 4.1, Output RPI 20 ms)
            ManSL02 : vendor 1 type 35 code 16 (PointIO 2, rev 1.1, Input RPI 10 ms, Output RPI 20 ms)
            ManSL01 : vendor 1 type 35 code 16 (PointIO 1, rev 1.1, Input RPI 10 ms, Output RPI 20 ms)
                 Manifold_N058:1:O.Pt00Data   // Cell 1 Hold Back Stop Extended
                 Manifold_N058:1:O.Pt02Data   // Cell 1 Robot Stop Extended
         Conv_N053 : 1734-AENTR (Ethernet 192.168.1.53, rev 4.1, Output RPI 20 ms)
            ConvSL03 : 1734-IB8 (PointIO 3, rev 3.1)
            ConvSL04 : 1734-OB8E (PointIO 4, rev 3.1)
            ConvSL02 : vendor 1 type 35 code 16 (PointIO 2, rev 1.1, Input RPI 10 ms, Output RPI 20 ms)
            ConvSL01 : vendor 1 type 35 code 15 (PointIO 1, rev 1.2, Input RPI 10 ms, Output RPI 20 ms)
         C2_N021 : 1734-AENTR (Ethernet 192.168.1.21, rev 4.1, Output RPI 20 ms)
              C2_N021:O.Data[7].1   // Switch on CNC 3
              C2_N021:O.Data[7].3   // Switch on CNC 4
            C2SL06 : 1734-IB8 (PointIO 6, rev 3.1)
            C2SL07 : 1734-OB8E (PointIO 7, rev 3.1)
            C2SL05 : vendor 1 type 35 code 16 (PointIO 5, rev 1.1, Input RPI 10 ms, Output RPI 20 ms)
            C2SL04 : vendor 1 type 35 code 15 (PointIO 4, rev 1.2, Input RPI 10 ms, Output RPI 20 ms)
            C2SL02 : vendor 1 type 35 code 15 (PointIO 2, rev 1.2, Input RPI 10 ms, Output RPI 20 ms)
            C2SL01 : vendor 1 type 35 code 15 (PointIO 1, rev 1.2, Input RPI 10 ms, Output RPI 20 ms)
            C2SL03 : vendor 1 type 35 code 15 (PointIO 3, rev 1.2, Input RPI 10 ms, Output RPI 20 ms)
         C3_N031 : 1734-AENTR (Ethernet 192.168.1.31, rev 4.1, Output RPI 20 ms)
            C3SL05 : 1734-IB8 (PointIO 5, rev 3.1)
            C3SL06 : 1734-OB8E (PointIO 6, rev 3.1)
            C3SL04 : vendor 1 type 35 code 16 (PointIO 4, rev 1.1, Input RPI 10 ms, Output RPI 20 ms)
            C3SL03 : vendor 1 type 35 code 15 (PointIO 3, rev 1.2, Input RPI 10 ms, Output RPI 20 ms)
            C3SL01 : vendor 1 type 35 code 15 (PointIO 1, rev 1.2, Input RPI 10 ms, Output RPI 20 ms)
            C3SL02 : vendor 1 type 35 code 15 (PointIO 2, rev 1.2, Input RPI 10 ms, Output RPI 20 ms)
      @fcc730f7@:Partner : vendor 1 type 14 code 146 (ICP 1, rev 28.12)
END_MODULES

TYPE ABB_Cell :
STRUCT
   GoodParts : COUNTER;   // Good part total
   RejectedParts : COUNTER;   // Rejected part total
   PartEntering : BOOL;   // Part in transit from hold back to robot stop
END_STRUCT
END_TYPE

TYPE ABB_Cell_Safe :
STRUCT
   Perim : Cell_Perimeter;   // Cell Perimeter I/O
END_STRUCT
END_TYPE

TYPE AcceptResponse :
STRUCT
   Instance : DINT;
   Addr : SocketAddress;
END_STRUCT
END_TYPE

TYPE Cell_Perimeter :   // Cell Perimeter Safeties
STRUCT
   ConnStat : CONNECTION_STATUS;
   GateSW_Ch1 : BOOL;   // Gate Switch Ch1
   GateSW_Ch2 : BOOL;   // Gate Switch Ch2
   Ent_LC_Ch1 : BOOL;   // Entry Light Screen Ch1
   Ent_LC_Ch2 : BOOL;   // Entry Light Screen Ch2
   Exit_LC_Ch1 : BOOL;   // Exit Light Screen Ch1
   Exit_LC_Ch2 : BOOL;   // Exit Light Screen Ch2
   Ent_Mute1 : BOOL;   // Entry Mute 1 (Mute Signals Inverted)
   Ent_Mute2 : BOOL;   // Entry Mute 2 (Mute Signals Inverted)
   Exit_Mute1 : BOOL;   // Exit Mute 1 (Mute Signals Inverted)
   Exit_Mute2 : BOOL;   // Entry Mute 1 (Mute Signals Inverted)
   Ent_LC_Over : BOOL;   // Override Entry LC Muting
   Exit_LC_Over : BOOL;   // Override Exit LC Muting
   EntMuteStatOK : BOOL;   // Status of connection to muting sensors is OK
   ExitMuteStatOK : BOOL;   // Status of connection to muting sensors is OK
   OK : BOOL;   // Perimeter is Secure
   Ent_LC_Not_Blocked : BOOL;   // Inverted LCB bit
   Exit_LC_Not_Blocked : BOOL;   // Inverted LCB bit
END_STRUCT
END_TYPE

TYPE CNC_Datablock :   // Block of data to be exchanged between CNC and Cell
STRUCT
   Bools : DINT;   // 32 user defined bools to be used as needed for interlocks
   UserDef01 : DINT;   // User defined Dint 1
   UserDef02 : DINT;   // User defined Dint 2
   UserDef03 : DINT;   // User defined Dint 3
   UserDef04 : DINT;   // User defined Dint 4
   UserDef05 : DINT;   // User defined Dint 5
END_STRUCT
END_TYPE

TYPE CNC_Interlock :   // Data to be passed to and from CNCs to Main Cell
STRUCT
   ToCell : CNC_Datablock;   // Data block sent to the Cell from the CNC
   ToCNC : CNC_Datablock;   // Data block sent to the CNC from the Cell
END_STRUCT
END_TYPE

TYPE CNC_Safetys :   // Safety I/O on Mills
STRUCT
   ConnStat : CONNECTION_STATUS;
   LC_Ch1 : BOOL;   // CNC Entry Light Screen Channel 1
   LC_Ch2 : BOOL;   // CNC Entry Light Screen Channel 2
   DoorSW_Ch1 : BOOL;   // CNC Door Switch Channel 1
   DoorSW_Ch2 : BOOL;   // CNC Door Switch Channel 2
   EStop_Ch1 : BOOL;   // CNC E-Stop Button Channel 1
   EStop_Ch2 : BOOL;   // CNC E-Stop Button Channel 2
   UserDef1 : BOOL;   // Spare Channel 1
   UserDef2 : BOOL;   // Spare Channel 2
END_STRUCT
END_TYPE

TYPE Fanuc_Cell :
STRUCT
   GoodParts : COUNTER;   // Good part total
   RejectedParts : COUNTER;   // Rejected part total
   PartEntering : BOOL;   // Part in transit from hold back to robot stop
   Mill_A : Mill_Data;
   Mill_B : Mill_Data;
END_STRUCT
END_TYPE

TYPE Fanuc_Cell_Safe :   // Data related to Fanuc Machining Cell
STRUCT
   ConnStat : CONNECTION_STATUS;
   CNC_A : CNC_Safetys;   // First CNC
   CNC_B : CNC_Safetys;   // Second CNC
   Perim : Cell_Perimeter;   // Cell Perimeter I/O
END_STRUCT
END_TYPE

TYPE Mill_Data :
STRUCT
   GoodParts : COUNTER;   // Good part total
   RejectedParts : COUNTER;   // Rejected part total
   PartEntering : BOOL;   // Part in transit from hold back to robot stop
END_STRUCT
END_TYPE

TYPE Mill_Safetys :   // Safety I/O on Mills
STRUCT
   LC_Ch1 : BOOL;   // Mill Entry Light Screen Channel 1
   LC_Ch2 : BOOL;   // Mill Entry Light Screen Channel 2
   DoorSW_Ch1 : BOOL;   // Mill Door Switch Channel 1
   DoorSW_Ch2 : BOOL;   // Mill Door Switch Channel 2
END_STRUCT
END_TYPE

TYPE OpenConnParams :
STRUCT
   Timeout : DINT;
   DestAddr : STRING;
END_STRUCT
END_TYPE

TYPE P_DescList :   // Code / Description List Entry
STRUCT
   Code : DINT;   // Code for which to look up Description
   Desc : STRING_40;   // Description for given Code
END_STRUCT
END_TYPE

TYPE P_PF52x_Inp :   // PF523 and PF525 Input Assembly
STRUCT
   DriveStatus : INT;
   DriveStatus_Ready : BOOL;
   DriveStatus_Active : BOOL;
   DriveStatus_CommandDir : BOOL;
   DriveStatus_ActualDir : BOOL;
   DriveStatus_Accelerating : BOOL;
   DriveStatus_Decelerating : BOOL;
   DriveStatus_Faulted : BOOL;
   DriveStatus_AtReference : BOOL;
   DriveStatus_CommFreqCnt : BOOL;
   DriveStatus_CommLogicCnt : BOOL;
   DriveStatus_ParmsLocked : BOOL;
   DriveStatus_DigIn1Active : BOOL;
   DriveStatus_DigIn2Active : BOOL;
   DriveStatus_DigIn3Active : BOOL;
   DriveStatus_DigIn4Active : BOOL;
   OutputFreq : INT;
   Fault1Code : INT;
   OutputCurrent : INT;
   OutputPower : INT;
END_STRUCT
END_TYPE

TYPE P_PF52x_Out :   // PF523 and PF525 Output Assembly
STRUCT
   LogicCommand : INT;
   LogicCommand_Stop : BOOL;
   LogicCommand_Start : BOOL;
   LogicCommand_Jog : BOOL;
   LogicCommand_ClearFaults : BOOL;
   LogicCommand_Forward : BOOL;
   LogicCommand_Reverse : BOOL;
   LogicCommand_ForceKeypadCtrl : BOOL;
   LogicCommand_MOPIncrement : BOOL;
   LogicCommand_AccelTime1 : BOOL;
   LogicCommand_AccelTime2 : BOOL;
   LogicCommand_DecelTime1 : BOOL;
   LogicCommand_DecelTime2 : BOOL;
   LogicCommand_SpdRefSel0 : BOOL;
   LogicCommand_SpdRefSel1 : BOOL;
   LogicCommand_SpdRefSel2 : BOOL;
   LogicCommand_MOPDecrement : BOOL;
   FreqCommand : INT;
END_STRUCT
END_TYPE

TYPE PalletStop :
STRUCT
   Ext : BOOL;   // Extend Stop
   Ret : BOOL;   // Retract Stop
END_STRUCT
END_TYPE

TYPE SocketAddress :
STRUCT
   Family : INT;
   Port : INT;
   Addr : DINT;
END_STRUCT
END_TYPE

TYPE STRING_12 :
STRUCT
   LEN : DINT;
   DATA : SINT[12];
END_STRUCT
END_TYPE

TYPE STRING_16 :
STRUCT
   LEN : DINT;
   DATA : SINT[16];
END_STRUCT
END_TYPE

TYPE STRING_20 :
STRUCT
   LEN : DINT;
   DATA : SINT[20];
END_STRUCT
END_TYPE

TYPE STRING_40 :
STRUCT
   LEN : DINT;
   DATA : SINT[40];
END_STRUCT
END_TYPE

TYPE STRING_8 :
STRUCT
   LEN : DINT;
   DATA : SINT[8];
END_STRUCT
END_TYPE

ADD_ON_INSTRUCTION P_Alarm   (* revision 3.1 00 Release, vendor Rockwell Automation, ExecutePrescan, ExecuteEnableInFalse *)
// Alarm
// Revision note:
// See Release Notes for Library 3.1-xx for details. Added Maintenace Test command, changed severity ranges and names to match FTAE (for linking to FTView 8).
// Help:
// Copyright © Rockwell Automation, Inc.  All Rights Reserved.
// This instruction monitors one input condition and provides one Alarm with:
//   * configurable latching (reset required) and acknowledgement requirement
//   * configurable alarm severity
//       1 = Low  (blue, typ. informational)
//       2 = Medium  (yelllow, typ. warning)
//       3 = High  (red, typ. process exception)
//       4 = Highest  (magenta, typ. equip. fault)
//   * configurable minimum ON time (e.g., to ensure it is seen by the HMI)
//   * commands to suppress/unsuppress (Prog), shelve/unshelve (Oper)
//         and disable/enable (Maint) the alarm.
//   * configurable amount of time shelved to automatically unshelve an alarm
//   * FTA&E support for suppressed, shelved and disabled states (V7.0)
//   * A Maintenance "Test" command, which triggers the alarm for the minimum
//      alarm time for testing purposes.
// NOTE regarding parameter naming:
//   FTAE names (same as ALMD instruction) are used instead
//   of the ANSI/ISA 18.2-2009 names, as follows:
//    "Disabled" is the equivalent of "Out of Service" in ISA 18.2.
//       (The Disabled state is owned by Maintenance.)
//    "Suppressed" is the equivalent of "Suppressed by Design" in
//       ISA 18.2. (The Suppressed state is owned by Program logic.)
//    "Shelved" is the same as in ISA 18.2.
//       (The Shelved state is owned by Operator, but may be cleared
//       by Program logic based on time, shift change, etc.)
// This instruction is usually nested within other instructions, with one instance
// used for each Alarm generated by the containing instruction.  It may also be
// used as a standalone instruction for Alarm conditions generated by custom logic.
// FTAE Alarm Setup:
//   (object).(alarm).Com_AE.0:  Alarm to FTAE
//     .Com_AE.1:   Ack to/from FTAE
//     .Com_AE.3:   Shelved from FTAE Status
//     .Com_AE.4:   Shelve/Reshelve to FTAE Control (auto reset)
//     .Com_AE.5:   Unshelve to FTAE Control (auto reset)
//     .Com_AE.6:   Suppressed to/from FTAE
//     .Com_AE.8:   Unsuppress to FTAE Control (auto reset)
//     .Com_AE.9:   Disabled to/from FTAE
//     .Com_AE.11: Enable to FTAE Control (auto reset)
//    all other bits unused
//     .Cfg_MaxShelfT is also used in FTAE config.
VAR_INPUT
   Inp : BOOL := 1; {visible}   // Alarm Condition Input 1=Alarm
   Inp_Reset : BOOL; {visible}   // 1=Reset Alarm requiring reset
   Cfg_Exists : BOOL := 1;   // 1=Alarm configured to exist, 0=Does not exist, don't scan
   Cfg_ResetReqd : BOOL;   // 1=Latched Alarm, a Reset is required to clear this Alarm
   Cfg_AckReqd : BOOL := 1;   // 1=Acknowledge required for this Alarm
   Cfg_AllowShelve : BOOL := 1;   // 1=Allow Operator to Shelve this Alarm
   Cfg_AllowDisable : BOOL := 1;   // 1=Allow Maintenance to Disable this Alarm
   Cfg_PCmdClear : BOOL := 1;   // 1=Clear Program Commands on receipt 0=Leave Set
   Cfg_Severity : INT := 750;   // Alarm Severity: 1..250=Low, 251..500=Medium, 501..750=High, 751..1000=Urgent
   Cfg_AlmMinOnT : DINT := 5;   // Minimum time Alm output stays on (sec)
   Cfg_MaxShelfT : INT := 480;   // Auto unshelve after shelved this long (1..32767 minutes)
   PCfg_AllowExist : BOOL := 1;   // 1=Alarm can be configured to exist, 0=other configs make alarm meaningless
   PCmd_Reset : BOOL;   // Program Command to Reset latched alarm
   PCmd_Ack : BOOL;   // Program Command to Acknowledge alarm
   PCmd_Suppress : BOOL;   // Program Command to Suppress by Design (inhibits new alarm)
   PCmd_Unsuppress : BOOL;   // Program Command to Unsuppress (allows new alarm)
   PCmd_Unshelve : BOOL;   // Program Command to Unshelve (e.g., on shift change)
   OCmd_Reset : BOOL;   // Operator Command to Reset latched alarm
   OCmd_Ack : BOOL;   // Operator Command to Acknowledge alarm
   OCmd_Shelve : BOOL;   // Operator Command to Shelve Alarm (inhibits new alarm)
   OCmd_Unshelve : BOOL;   // Operator Command to Unshelve alarm (allows new alarm)
   MCmd_Disable : BOOL;   // Maintenance Command to Disable alarm (inhibits new alarm)
   MCmd_Enable : BOOL;   // Maintenance Command to Enable alarm (allows new alarm)
   MCmd_Test : BOOL;   // Maintenance Command to Test alarm (issued for minimum alarm time)
END_VAR
VAR_OUTPUT
   Val_Notify : SINT; {access Read Only}   // Current Alarm Severity and Acknowledgement (enumeration)
   Val_MinToUnshelve : DINT; {access Read Only, visible}   // Number of minutes until this alarm unshelves itself (mmm:ss)
   Val_SecToUnshelve : DINT; {access Read Only, visible}   // Number of Seconds until this alarm unshelves itself (mmm:ss)
   Alm : ALIAS FOR Com_AE.0; {visible}   // Alarm output 1=In Alarm
   Ack : ALIAS FOR Com_AE.1; {visible}   // Alarm acknowledged status: 1=Ack rcvd
   Shelved : ALIAS FOR Com_AE.3; {visible}   // 1=Alarm has been Shelved by Operator (inhibits new alarm)
   Suppressed : ALIAS FOR Com_AE.6; {visible}   // 1=Alarm has been Suppressed by Program (inhibits new alarm)
   Disabled : ALIAS FOR Com_AE.9; {visible}   // 1=Alarm has been Disabled by Maintanance (inhibits new alarm)
   Sts_AlmInh : BOOL; {access Read Only}   // 1=Alarm has been suppressed, shelved or disabled, display "I" icon
   Sts_Err : BOOL; {access Read Only}   // 1=Error in Config: see detail Err_ bits for reason
   Err_Timer : BOOL; {access Read Only}   // 1=Error in Config: Alarm Min On Time, Shelf Time (use 0 to 2147483)
   Err_Severity : BOOL; {access Read Only}   // 1=Error in Config: Invalid Severity (use 1 to 4)
   Rdy_Reset : BOOL; {access Read Only}   // Ready to receive OCmd_Reset (enables button)
   Rdy_Ack : BOOL; {access Read Only}   // Ready to receive OCmd_Ack (enables button)
   Rdy_Shelve : BOOL; {access Read Only}   // Ready to receive OCmd_Shelve (enables button)
   Rdy_Unshelve : BOOL; {access Read Only}   // Ready to receive OCmd_Unshelve (enables button)
   Rdy_Disable : BOOL; {access Read Only}   // Ready to receive MCmd_Disable (enables button)
   Rdy_Enable : BOOL; {access Read Only}   // Ready to receive MCmd_Enable (enables button)
   Rdy_Test : BOOL; {access Read Only}   // Ready to receive MCmd_Test (enables button)
   P_Alarm : BOOL;   // Unique Parameter Name for auto - discovery
END_VAR
VAR
   Wrk_Alm : BOOL; {access None}   // Internal Alarm Status
   Wrk_Suppressed : BOOL; {access None}   // Internal Alarm Suppressed Status
   Wrk_AlmMinOnT : TIMER := (PRE := 5000); {access None}   // Alarm output minimum ON time to be seen by alarm server
   Wrk_AutoAckT : TIMER := (PRE := 5000); {access None}   // Time to clear Ack bit when Ack not required
   Wrk_ShelfT : TIMER; {access None}   // Time to auto Unshelve a Shelved Alarm
   Inf_Tab : SINT;   // Tab to display (FTView ME)
   Com_AE : INT := 2#0000_0000_0000_0010;   // Communication with HMI / Alarm/Event Server (see bit descriptions)
        .1   // Acked from AE Status, Ack to AE Control
        .10   // (not used)
        .11   // Enable to AE Control
        .12   // (not used)
        .13   // (not used)
        .14   // (not used)
        .15   // (not used)
        .2   // (not used)
        .3   // Shelved from AE Status
        .4   // Shelve to AE Control
        .5   // Unshelve to AE Control
        .6   // Suppressed from AE Status, Suppress to AE Control
        .7   // (not used)
        .8   // Unsuppress to AE Control
        .9   // Disabled from AE Status, Disable to AE Control
        .0   // Alarm to AE
   Cfg_Tag : STRING_20 := 'P_Alarm';   // Alarm Tag Text (e.g., "LAHH-101")
   Cfg_Cond : STRING_20 := 'Alarm Condition';   // Alarm Condition Text (e.g., "High-High PV")
   Wrk_SecToUnshelve : DINT; {access None}   // Number of seconds until this alarm unshelves itself
   Inf_Lib : STRING_12 := 'RA-BAS'; {access Read Only}   // Display Library for Faceplate call-up
   Inf_Type : STRING_16 := 'P_Alarm'; {access Read Only}   // Must contain AOI name, used for HMI and Information S/W
END_VAR
